(* IEC 61131-3 sources: codesys-mcp-toolkit/standalone-sync/sources_st/511_05, 13 files *)

(* ---- CLIENT_STATE.dut.st ---- *)
// @OBJECT_ID: 38106bf3-2e28-4407-a341-929dcc35d1f5
// @DECLARATION
// шаг состояния клиента
{attribute 'strict'}
TYPE CLIENT_STATE :
(
	CREATE	:=	 0,
	WAITING	:=	10,
	SEND	:=	20,
	RECEIVE :=  30
);
END_TYPE

(* ---- Coils.dut.st ---- *)
// @OBJECT_ID: 733d5e5a-4ad1-4a84-973a-cf97214e756a
// @DECLARATION
{attribute 'pack_mode' := '1'}
TYPE Coils :
STRUCT
// --- Режимы работы (команды из HMI) ---
xManualMode_Diazo   : BOOL;        // 1. Ручной режим Diazo
xManualMode_Soda    : BOOL;        // 2. Ручной режим Soda
xManualMode_Steam   : BOOL;        // 3. Ручной режим Steam
// --- Управление водой имитатором ---
xWaterValve_AutoMode : BOOL;       // 4. TRUE=Автоматический режим, FALSE=Ручной
xWaterValve_HmiOpen  : BOOL;       // 5. Открытие по кнопке из HMI (в ручном режиме)
xWaterValve_AutoReq  : BOOL;       // 6. Запрос на открытие от автоматики
// --- Сигналы запуска ---
xWaterStart          : BOOL;       // 7. Запуск дозы воды из HMI
xStartHeating_511    : BOOL;       // 8. Запуск прогрева
// --- Сигналы и статусы стадии промывки (Cascade Drain) ---
xStartCoupling_511   : BOOL;       // 9. Запуск с HMI: признак запуска стадии промывки
xCouplingActive_511  : BOOL;       // 10. Статус для HMI: признак "работа идет"
xCouplingDone_511    : BOOL;       // 11. Статус для HMI: признак "успешно готово"
// --- Режим удержания температуры ---
xKeepTempHeating_511 : BOOL;       // 12. TRUE = удержание температуры после нагрева, FALSE = разовый нагрев
// --- Служебные ---
PLC_READ             : BOOL := TRUE; // 13. Флаг чтения PLC
END_STRUCT
END_TYPE

(* ---- HoldingRegs.dut.st ---- *)
// @OBJECT_ID: e939cef4-c06c-4a02-a15a-aa924dd4400b
// @DECLARATION
{attribute 'pack_mode' := '4'}
TYPE HoldingRegs :
STRUCT
// =============================================================
// Модули M7–M9 (MDS AO-2UI) - Управление клапанами (Выходы 4-20мА)
// =============================================================

// --- Управление запорно-регулирующими клапанами (задание 0..100%) ---
AO1_CmdValveDiazo   : REAL;    // 101. Управление клапаном диазосоединения
AO2_CmdValveSoda    : REAL;    // 103. Управление клапаном едкого натра 14%
AO3_CmdValveSteam   : REAL;    // 105. Управление клапаном пара 6 ати

// --- Уставки с панели (ручной режим) ---
rValveManSet_Diazo  : REAL := 0.0;    // 107. Уставка с панели: Диазо
rValveManSet_Soda   : REAL := 0.0;    // 109. Уставка с панели: Сода
rValveManSet_Steam  : REAL := 0.0;    // 111. Уставка с панели: Пар

// --- Переменные для автоматического управления (выходы ПИД-регуляторов) ---
rAutoSet_Diazo      : REAL;           // 113. Выход ПИД расхода диазо
rAutoSet_Soda       : REAL;           // 115. Выход ПИД расхода соды
rAutoSet_Steam      : REAL;           // 117. Выход ПИД расхода пара

// --- Технологические уставки ---
rWaterDose          : REAL := 5.0;    // 119. Заданная доза воды, м³ (5 кубов)
rSetTempApp511      : REAL := 86.0;   // 121. Уставка температуры
rSetFlowDiazo_511   : REAL;           // 123. Уставка мгновенного расхода диазосоединения (до 19 м³/ч)
rSetPh_511          : REAL;           // 125. Целевая уставка pH (9.5..12 ед.)

// --- Настройки алгоритма опустошения емкости (для наладчика) ---
rZeroFlowThreshold_511 : REAL := 0.2; // 127. Порог падения расхода диазо (м³/ч), ниже которого считаем, что емкость пуста
uiEmptyDelaySec_511    : UINT := 20;  // 129. Задержка фиксации пустого трубопровода (сек)

// --- Настройки ПИД-регуляторов (для наладки контуров с HMI) ---
rKp_Diazo_511        : REAL := 1.0;   // 131. Пропорциональный коэффициент контура расхода диазосоединения
rTn_Diazo_511        : REAL := 5.0;   // 133. Время интегрирования контура расхода диазосоединения (сек)
rKp_pH_511           : REAL := 2.0;   // 135. Пропорциональный коэффициент контура pH
rTn_pH_511           : REAL := 10.0;  // 137. Время интегрирования контура pH (сек)
rKp_Steam_511        : REAL := 2.0;   // 139. Пропорциональный коэффициент контура пара (нагрева)
rTn_Steam_511        : REAL := 15.0;  // 141. Время интегрирования контура пара (сек)
rTv_Steam_511        : REAL := 0.0;   // 143. Время дифференцирования контура пара (сек)

END_STRUCT
END_TYPE

(* ---- InputRegs.dut.st ---- *)
// @OBJECT_ID: e329769f-e235-4ed6-8989-e7d305dd0344
// @DECLARATION
{attribute 'pack_mode' := '4'}
TYPE InputRegs :
STRUCT
	COILS : DINT := 0;
	INPUTS: DINT := 0;
	HOLDINGS: DINT := 0;
	INPUTREGS: DINT := 0;

  // МОДУЛЬ АНАЛОГОВЫХ ВХОДОВ (AI)
  	{region M1_K3_AI_10_08_00 }
    // =========================================================================
    // Первые 3 канала: Сигнализация положений (% открытия) клапанов [1, 2]
    (* adr 9 *)  rPosValveDiazo  : REAL; // Канал 1: Обратная связь клапана диазосоединения
    (* adr 11 *) rPosValveSoda   : REAL; // Канал 2: Обратная связь клапана едкого натра 14%
    (* adr 13 *) rPosValveSteam  : REAL; // Канал 3: Обратная связь клапана пара

    // Канал 4: рН-метр
    (* adr 15 *) rPhApp511       : REAL; // Канал 4: Показания pH-метра аппарата 511 (диапазон 9,5..12 ед.)
			{endregion}

	{region M5_MDS_3RTD_1 }
	(* adr 17 *) rTempApp511     : REAL; // Температура в аппарате 511 (до 100 С°)

   	{endregion}

	{region tenzo tv006c }
	(* adr 19 *) WE_1            : REAL;
	(* adr 21 *) WE_2            : REAL;

   	{endregion}

	{region tenzo ELMER }

	(* adr 23 *) IR_FlowSoda   : REAL; // Текущий расход щелочи , л/мин (или м3/ч)
	(* adr 25 *) IR_TotalSoda   : REAL; // Накопленный объем щелочи, л (или м3)
	(* adr 27 *) IR_FlowWater     : REAL; // Текущий расход воды, л/мин (или м3/ч)
	(* adr 29 *) IR_TotalWater   : REAL; // Накопленный объем воды, л (или м3)

    // Выходные сигналы загрузки воды
	(* adr  31*)   rWaterLoaded   : REAL;    // Сколько воды загружено, м³
	(* adr 32*)    rWaterStatus   : REAL;    // Статус загрузки воды: 0=IDLE 1=RUNNING 2=DONE 3=ABORTED

	(* adr  33*)  IR_FlowDiazo   : REAL; // Текущий мгновенный расход диазосоединения (м3/ч) [3]
	(* adr  35*)  IR_TotalDiazo   : REAL; // Текущий расход диазосоединения, л/мин (или м3/ч)

	(* adr  37*)  rDizoStatus   : REAL; // Текущий расход диазосоединения, л/мин (или м3/ч)

	(* adr  39*) rDiazoLoaded   : REAL; // Текущий расход диазосоединения, л/мин (или м3/ч)
rTimeLeft_511:REAL ;///Оставшиеся секунды при падении расхода
	 rStateCode_511:REAL;//

   	{endregion}

END_STRUCT
END_TYPE

(* ---- Inputs.dut.st ---- *)
// @OBJECT_ID: a5893dca-19fc-4f6d-bdfc-9d37b1592804
// @DECLARATION
{attribute 'pack_mode' := '1'}
TYPE Inputs :
STRUCT
			// =============================================================
			// Модуль M11 (MDS DIO-16BD) - Статусы насосов (Дискретные входы)
			// =============================================================
			{region M11 - MDS DIO-16BD (Статусы насосов)}

    // Выходная переменная на физическое реле/соленоид
    xWaterValve_Out     : BOOL;  // 1 канал ФЕ
	xWaterValve_SQH :BOOL;
	xWaterValve_SQL   :BOOL;
			{endregion}
END_STRUCT
END_TYPE

(* ---- GVL.gvl.st ---- *)
// @OBJECT_ID: 3f8320a4-dc77-4c55-9b52-3e7e3f19e8e0
// @DECLARATION
{attribute 'qualified_only'}

VAR_GLOBAL

	gInputRegs	:	InputRegs;
	gHoldingRegs	:	HoldingRegs;
	gInputs	:	Inputs;
	gCoils	:	Coils;
    // =========================================================================
    // АНАЛОГОВЫЕ ВХОДЫ (Опрос датчиков)
    // =========================================================================
    rPressPump207v      : REAL; // Давление насоса мембранного 207в (0.5..6 кгс/см2)
    rTempApp511         : REAL; // Температура реакционной среды в аппарате 511 (до 100 °C)
    rPhApp511           : REAL; // Показания pH-метра аппарата 511 (9.5..12 ед.)

	WE_1_s:WORD;
	WE_1_f:WORD;

	WE_2_s:WORD;
	WE_2_f:WORD;

	sStateStr_511:string(255);

    // =========================================================================
    // СЧЕТЧИКИ И РАСХОДОМЕРЫ (Опрос текущего расхода и накопленного объема)
    // =========================================================================
    rFlowDiazo          : REAL; // Текущий расход диазосоединения (м3/ч)
    rTotalDiazo         : REAL; // Накопленный объем диазосоединения (м3)

    rFlowSoda           : REAL; // Текущий расход едкого натра 14% (м3/ч)
    rTotalSoda          : REAL; // Накопленный объем едкого натра 14% (м3)

    rFlowWater          : REAL; // Текущий расход воды артезианской/деминерализованной (м3/ч)
    rTotalWater         : REAL; // Накопленный объем воды / счетчик дозы (м3)

    // =========================================================================
    // СИГНАЛЫ СОСТОЯНИЯ КЛАПАНОВ (Входы обратной связи)
    // =========================================================================
    rPosValveDiazo      : REAL; // Сигнализация положения (% открытия) клапана диазосоединения
    rPosValveSoda       : REAL; // Сигнализация положения (% открытия) клапана едкого натра
    rPosValveSteam      : REAL; // Сигнализация положения (% открытия) клапана пара

    xStsValveWaterOpen  : BOOL; // Сигнализатор положения отсечного пневмокрана воды - ОТКРЫТ
    xStsValveWaterClose : BOOL; // Сигнализатор положения отсечного пневмокрана воды - ЗАКРЫТ

    // =========================================================================
    // АНАЛОГОВЫЕ И ДИСКРЕТНЫЕ ВЫХОДЫ (Управление исполнительными механизмами)
    // =========================================================================
    rCmdValveDiazo  AT  %QW0    : WORD; // Управление регулирующим клапаном диазосоединения (0..100%)
    rCmdValveSoda   AT  %QW1    : WORD; // Управление регулирующим клапаном едкого натра (0..100%)
    rCmdValveSteam  AT  %QW2    : WORD; // Управление регулирующим клапаном пара для поддержания температуры (0..100%)
    xCmdValveWater      : BOOL; // Дискретное управление отсечным пневмокраном воды (закрытие при достижении дозы)

    // =========================================================================
    // ПЕРЕМЕННЫЕ HMI / СЕНСОРНОЙ ПАНЕЛИ (Уставки и задания)
    // =========================================================================
    rSpTempApp511       : REAL; // Задание поддерживаемой температуры в аппарате (до 100 °C)
    rSpFlowDiazo        : REAL; // Задание необходимого расхода диазосоединения (до 19 м3/ч)
    rSpFlowSoda         : REAL; // Задание необходимого расхода едкого натра (до 7.35 м3/ч)
    rSpDoseWater        : REAL; // Задание необходимой дозы воды (до 7.35 м3/ч)

    // Переменные для алгоритма дозирования щелочи
    rSpPhLow            : REAL := 9.2; // Нижний порог pH для увеличения открытия клапана щелочи
    rSpPhHigh           : REAL := 9.7; // Верхний порог pH для уменьшения открытия клапана щелочи
    rSpPhTargetMatch    : REAL := 9.6; // Порог pH для открытия клапана щелочи на стадии "сочетания"
    rSpPhTargetClose    : REAL := 9.5; // Порог pH для закрытия клапана щелочи
MDS_3RTD_1_start_ad : POINTER TO ARRAY[0..10] OF WORD;;
END_VAR

(* ---- PVL.gvl.st ---- *)
// @OBJECT_ID: d4c88051-2adb-4578-9e31-dd205f936f9c
// @DECLARATION
{attribute 'qualified_only'}
VAR_GLOBAL PERSISTENT RETAIN
	rHoldingRegs: HoldingRegs;
END_VAR

(* ---- FC_Write_AO.func.st ---- *)
// @OBJECT_ID: 58eab0a1-f642-4bbd-ba35-3845d9d3886b
// @DECLARATION
FUNCTION FC_Write_AO : BOOL
VAR_INPUT
    VAL_IN  : REAL;    // Входное значение (например, от ПИД 0..1000)

    pOutput : POINTER TO ARRAY[0..1] OF WORD; // Адрес физических регистров модуля
END_VAR
VAR
    TMP     : REAL;
    dwValue : DWORD;
	    X1      : REAL:=0;    // Мин. вход (например, 0)
    X2      : REAL:=100;    // Макс. вход (например, 1000)
    Y1      : REAL:=4;    // Мин. ток (например, 4.0)
    Y2      : REAL:=20;    // Макс. ток (например, 20.0)
END_VAR

// @IMPLEMENTATION

// 1. Проверка на нулевой указатель и деление на ноль
IF pOutput = 0 OR (X2 = X1) THEN
    FC_Write_AO := FALSE;
    RETURN;
END_IF;

// 2. Линейное масштабирование (из входного диапазона в 4..20мА)
TMP := (Y2 - Y1) / (X2 - X1) * (VAL_IN - X1) + Y1;

// 3. Преобразование REAL во внутреннее битовое представление DWORD
dwValue := OSCAT_BASIC.REAL_TO_DW(TMP);

// 4. Запись напрямую в память по указателю (разбивка на 2 WORD)
// В ПЛК Абак обычно старшее слово идет первым (зависит от настроек модуля)
pOutput^[0] := OSCAT_BASIC.WORD_OF_DWORD(dwValue, 1); // High Word
pOutput^[1] := OSCAT_BASIC.WORD_OF_DWORD(dwValue, 0); // Low Word

FC_Write_AO := TRUE;

(* ---- FC_Write_AO_CDAB.func.st ---- *)
// @OBJECT_ID: c5f4f6d9-aef8-4f24-80c9-f3d975bafcdd
// @DECLARATION
FUNCTION FC_Write_AO_CDAB : BOOL
VAR_INPUT
    rValIn   : REAL;    // Входная уставка (0..100)
    pOutput  : POINTER TO ARRAY[0..1] OF WORD;
    rInMin   : REAL;
    rInMax   : REAL;
    rOutMin  : REAL;
    rOutMax  : REAL;
END_VAR
VAR
    rScaled  : REAL;
    dwRaw    : DWORD;
	dwCDAB: DWORD;
    pReal    : POINTER TO DWORD;
END_VAR

// @IMPLEMENTATION
// 1. Линейное масштабирование (Scale)
// Формула: Out = ((In - InMin) * (OutMax - OutMin) / (InMax - InMin)) + OutMin
IF (rInMax <> rInMin) THEN
    rScaled := ((rValIn - rInMin) * (rOutMax - rOutMin) / (rInMax - rInMin)) + rOutMin;
ELSE
    rScaled := rOutMin;
END_IF

// 2. Получаем битовое представление REAL как DWORD
pReal := ADR(rScaled);
dwRaw := pReal^;

// 3. Перепаковка в формат CDAB
// Исходный (ABCD): [Byte3][Byte2][Byte1][Byte0]
// Формат CDAB:     [Byte1][Byte0][Byte3][Byte2]
// То есть меняем местами слова (WORD)

dwCDAB := ROL(dwRaw, 16); // Простейший способ поменять слова местами

// 4. Запись результата по указателю
IF pOutput <> 0 THEN
    pOutput^[1] := DWORD_TO_WORD(dwCDAB AND 16#FFFF);        // Младшее слово CDAB (бывшее старшее AB)
    pOutput^[0] := DWORD_TO_WORD(SHR(dwCDAB, 16));           // Старшее слово CDAB (бывшее младшее CD)
    FC_Write_AO_CDAB := TRUE;
ELSE
    FC_Write_AO_CDAB := FALSE;
END_IF

(* ---- FB_AI.fb.st ---- *)
// @OBJECT_ID: 3f0a8be8-2f33-46cf-a2ab-090e0d72fc51
// @DECLARATION
FUNCTION_BLOCK FB_AI
VAR_INPUT
	F_WORD_IN : WORD;
	S_WORD_IN : WORD;
	X1 : REAL:=4;
	Y1 : REAL:=0;
	X2 : REAL:=20;
	Y2 : REAL:=100;
	RANGE_CONV:BOOL:=TRUE;
END_VAR
VAR
	TMP:REAL;
END_VAR
VAR_OUTPUT
	VAL_OUT : REAL;
END_VAR

// @IMPLEMENTATION
TMP := OSCAT_BASIC.DW_TO_REAL(X:= OSCAT_BASIC.DWORD_OF_WORD(W1:= F_WORD_IN , W0:= S_WORD_IN ));
IF (RANGE_CONV)
THEN
	IF (TMP=9999 OR TMP=-9999 OR TMP=-7777 OR TMP=7777)
	THEN
		VAL_OUT :=  TMP;
	ELSE
		VAL_OUT :=  (Y2 - Y1) / (X2 - X1) * (TMP - X1) + Y1;
	END_IF

ELSE
	VAL_OUT :=  TMP;
END_IF

(* ---- FB_ModbusToFloatArray.fb.st ---- *)
// @OBJECT_ID: 8d81ca1b-e4d0-4e94-b201-9038cef709f6
// @DECLARATION
FUNCTION_BLOCK FB_ModbusToFloatArray
VAR_INPUT
    aDataIn : ARRAY [0..219] OF WORD; // Входной массив (до 120 регистров)
    iQty    : INT := 1;               // Количество FLOAT переменных для обработки (макс 60)
    iMode   : INT := 1;               // Режим: 0=1234, 1=3412 (частый), 2=2143, 3=4321
END_VAR
VAR_OUTPUT
    aDataOut : ARRAY [0..119] OF REAL; // Выходной массив
    xError   : BOOL;                  // Флаг ошибки (если iQty > 60)
END_VAR
VAR
    i : INT;
    uConverter : U_WordToReal;
    wLow : WORD;
    wHigh : WORD;
    wTemp1 : WORD;
    wTemp2 : WORD;
END_VAR

// @IMPLEMENTATION

// Сброс ошибки
xError := FALSE;

// Защита от выхода за пределы массива
IF iQty < 1 OR iQty > 120 THEN
    xError := TRUE;
    RETURN;
END_IF

// Основной цикл
FOR i := 0 TO (iQty - 1) DO

    // Получаем пару регистров из массива
    // i*2 - это начало пары (0, 2, 4...)
    wTemp1 := aDataIn[i * 2];     // Первый регистр пары
    wTemp2 := aDataIn[(i * 2) + 1]; // Второй регистр пары

    CASE iMode OF
        // ---------------------------------------------------------
        // Mode 0: 1234 (Big Endian)
        // Порядок: [HighWord] [LowWord]
        // ---------------------------------------------------------
        0:
            wHigh := wTemp1;
            wLow  := wTemp2;

        // ---------------------------------------------------------
        // Mode 1: 3412 (Middle Little / Word Swap) -> САМЫЙ ЧАСТЫЙ для Modbus
        // Порядок: [LowWord] [HighWord]
        // Регистры меняются местами, байты внутри - нет.
        // ---------------------------------------------------------
        1:
            wHigh := wTemp2;
            wLow  := wTemp1;

        // ---------------------------------------------------------
        // Mode 2: 2143 (Middle Big / Byte Swap)
        // Порядок: [HighWord swapped] [LowWord swapped]
        // Байты меняются местами внутри каждого слова.
        // ---------------------------------------------------------
        2:
            wHigh := ROL(wTemp1, 8); // Меняем байты местами
            wLow  := ROL(wTemp2, 8);

        // ---------------------------------------------------------
        // Mode 3: 4321 (Little Endian)
        // Порядок: [LowWord swapped] [HighWord swapped]
        // Полный разворот: меняются и слова, и байты.
        // ---------------------------------------------------------
        3:
            wHigh := ROL(wTemp2, 8);
            wLow  := ROL(wTemp1, 8);

        ELSE
            // По умолчанию используем 3412 (как самый популярный)
            wHigh := wTemp2;
            wLow  := wTemp1;
    END_CASE

    // Сборка DWORD из двух слов
    // Сдвигаем старшее слово на 16 бит влево и добавляем младшее
    uConverter.dwValue := SHL(WORD_TO_DWORD(wHigh), 16) OR WORD_TO_DWORD(wLow);

    // Запись результата в выходной массив
    aDataOut[i] := uConverter.rValue;

END_FOR

(* ---- ASK_prg.prg.st ---- *)
// @OBJECT_ID: 34a98575-253b-42d3-9455-2cb10a7687ff
// @DECLARATION
PROGRAM ASK_prg
VAR
Exatract:	FB_ModbusToFloatArray;
pt : POINTER TO  ARRAY [0..5] OF WORD  ;

//M1_K3_AI_10_08_00 AT %IW58: ARRAY [0..7] OF WORD ;

buff_abak: ARRAY [0..219] OF WORD ;
buff_MDS: ARRAY [0..219] OF WORD ;
buffR_1: ARRAY [0..119] OF REAL ;
start_ad_mds3rtd:INT:=0;
swap_mds3rtd:INT:=6;
start_ad_mds_8UId:INT:=18;
swap_mds_8UI:INT:=16;

AI: FB_AI;

	Info : __SYSTEM.VAR_INFO;

    pAddress : POINTER TO BYTE;
	adress:UDINT;
END_VAR

// @IMPLEMENTATION
//берем  с модуля  M1_K3_AI_10_08_00 значения  и  копируем в промежуточный буфер
SysMemCpy(ADR(buff_abak), ADR( %IW0), 8 * SIZEOF(WORD));

//берем  с модуля  MDS_3RTD_1  значения  и  копируем в промежуточный буфер
SysMemCpy(ADR(buff_MDS), ADR( %IW57), 6 * SIZEOF(WORD));

//берем  с  терминала  tv 006
SysMemCpy(ADR(buff_MDS[swap_mds3rtd]), ADR( %IW53), 2* SIZEOF(WORD));

//берем  с  терминала  tv 006
SysMemCpy(ADR(buff_MDS[swap_mds3rtd+2]), ADR( %IW55), 2* SIZEOF(WORD));

Exatract(aDataIn:=buff_MDS,aDataOut=>buffR_1,IQty:=65,iMode:=1);

// 3. Маппинг (Присвоение значений переменным структуры)
// -------------------------------------------------------------

// === Модуль M1 () ===
GVL.gInputRegs. rPosValveDiazo  := AIToFloat(buff_abak[0],0,100); //
GVL.gInputRegs.rPosValveSoda  := AIToFloat(buff_abak[1],0,100); //
GVL.gInputRegs.rPosValveSteam  := AIToFloat(buff_abak[2],0,100); //
GVL.gInputRegs.rPhApp511  := AIToFloat(buff_abak[4],0,14); //

// === Модуль M5 () ===

GVL.gInputRegs.rTempApp511  :=buffR_1[0];// TT 511
//GVL.gInputRegs.rTempApp511  :=FC_ModbusToRealSwapped(wWord1 := buff_MDS[0], wWord2 := buff_MDS[1]);
// === Модуль M2 () ===
GVL.rCmdValveDiazo := FloatToAI(gvl.gHoldingRegs.AO1_CmdValveDiazo);

GVL.rCmdValveSoda := FloatToAI(gvl.gHoldingRegs.AO2_CmdValveSoda);

GVL.rCmdValveSteam := FloatToAI(gvl.gHoldingRegs.AO3_CmdValveSteam);

// === Модуль M5 (Индексы 0..2) ===
//GVL.gInputRegs.rTempApp511   := buffR_1[0]; // TT 511

//// === весы  tenzo  M1 ===

	//AI(F_WORD_IN:= gvl.WE_1_f, S_WORD_IN:= gvl.WE_1_s, RANGE_CONV:=FALSE, VAL_OUT=> GVL.gInputRegs.WE_1);
GVL.gInputRegs.WE_1:=buffR_1[3];
GVL.gInputRegs.WE_2:=buffR_1[4];
//// === весы  tenzo  M2 ===
//AI(F_WORD_IN:= gvl.WE_2_f, S_WORD_IN:= gvl.WE_2_s, RANGE_CONV:=TRUE, VAL_OUT=> GVL.gInputRegs.WE_2);

(* ---- PLC_PRG.prg.st ---- *)
// @OBJECT_ID: 4c4237aa-22c6-43a4-ae1d-3ca0359860c2
// @DECLARATION
PROGRAM PLC_PRG // Antigravity Sync Test
VAR
    fbElemerREM         : fbElemerREM;

    (* Переменные из вкладки Modbus Generic Serial Slave I/O Mapping *)
    Hmi_Flow_Regs    AT %IW67  : ARRAY[0..1] OF WORD; (* Канал 0 (Мгновенный расход) *)
    Hmi_Volume_Regs  AT %IW63  : ARRAY[0..3] OF WORD; (* Канал 1 (Накопленный объем) *)
    xModbusCommError    : BOOL;                 (* Системный флаг ошибки связи с прибором *)
    xHmiResetCmd        : BOOL;                 (* Сигнал сброса сумматора с HMI-панели *)

    (* Выходные очищенные технологические переменные *)
    rCurrentFlowRate    : REAL;                 (* Мгновенный расход в систему, куб.м/ч *)
    lrAccumulatedVol    : LREAL;                (* Точный накопленный объем, куб.м *)
    sOperatorMessage    : STRING(255);          (* Сообщение для текстовой строки на панели *)

    fbWater             : FB_WaterLoading;      (* Наш исправленный ФБ дозирования *)

    // ============================================================
    // ПЕРЕМЕННЫЕ ДЛЯ ТЕСТИРОВАНИЯ И СИМУЛЯЦИИ СУММАТОРА
    // ============================================================
    xSimEnable          : BOOL := FALSE;        (* Включить режим симуляции (True = подмена датчиков) *)
    rSimFlowSpeed       : REAL := 20.0;         (* Скорость потока при открытом клапане, куб.м/ч *)
    rSimTotalStorage    : REAL := 125.45;       (* Внутренний виртуальный накопительный счетчик куб.м *)

    fbSimClock          : TON;                  (* Генератор тактов времени для подсчета объема *)
    rDeltaVolume        : REAL;                 (* Математический шаг приращения за 1 такт *)
    // ============================================================
END_VAR

// @IMPLEMENTATION
// ================================================================
// 1. ЧТЕНИЕ РЕАЛЬНЫХ ДАННЫХ ИЗ ПОЛЕВЫХ ПРИБОРОВ
// ================================================================
gvl.gInputRegs.IR_TotalSoda := F_ElemerREM_Volume(pBuf := ADR(%IW65));
gvl.gInputRegs.IR_FlowSoda  := F_ElemerREM_Flow(pBuf := ADR(%IW69));
gvl.gInputRegs.rTempApp511  := F_GetReal_BADC(pBuf := ADR(%IW57));

// ================================================================
// 2. ДИНАМИЧЕСКИЙ СИМУЛЯТОР РАСХОДОМЕРА ВОДЫ
// ================================================================
// Тактовый генератор: срабатывает каждые 100 мс (0.1 секунды) для плавности хода счета
fbSimClock(IN := xSimEnable AND NOT fbSimClock.Q, PT := T#100ms);

IF xSimEnable THEN
    // ЕСЛИ СИМУЛЯЦИЯ ВКЛЮЧЕНА:

    // Имитируем поведение потока в зависимости от команды на клапан
    IF gvl.gCoils.xWaterValve_AutoReq THEN
        // Клапан открыт автоматикой -> задаем симуляционный расход
        gvl.gInputRegs.IR_FlowWater := rSimFlowSpeed;

        // Расчет приращения сумматора за 100мс: (куб.м/ч * 0.1с) / 3600с
        IF fbSimClock.Q THEN
            rDeltaVolume := (rSimFlowSpeed * 0.1) / 3600.0;
            rSimTotalStorage := rSimTotalStorage + rDeltaVolume;
        END_IF;
    ELSE
        // Клапан закрыт -> поток прекращается
        gvl.gInputRegs.IR_FlowWater := 0.0;
    END_IF;

    // ПОДМЕНЯЕМ значение сумматора результатом симуляции для ФБ дозирования
    gvl.gInputRegs.IR_TotalWater := rSimTotalStorage;

ELSE
    // ЕСЛИ СИМУЛЯЦИЯ ВЫКЛЮЧЕНА (РАБОЧИЙ РЕЖИМ):

    // Читаем физический прибор с адреса %IW71 и %IW75
    gvl.gInputRegs.IR_TotalWater := F_ElemerREM_Volume(pBuf := ADR(%IW71));
    gvl.gInputRegs.IR_FlowWater  := F_ElemerREM_Flow(pBuf := ADR(%IW75));

    // Мягко синхронизируем симулятор, чтобы при включении тумблера счет не прыгал назад/вперед
    rSimTotalStorage := gvl.gInputRegs.IR_TotalWater;
END_IF;

// ================================================================
// 3. ВЫЗОВ И ПРОВЕРКА ФУНКЦИОНАЛЬНОГО БЛОКА ЗАГРУЗКИ ВОДЫ
// ================================================================
fbWater(
    rTotalVolume := gvl.gInputRegs.IR_TotalWater,        // Сюда идет либо физический объем, либо симуляция
    rDose        := gvl.gHoldingRegs.rWaterDose,         // Заданная уставка дозы (куб.м)
    rDeadband    := 0.05,                                // Упреждение закрытия (0.05 куб.м)
    xStart       := gvl.gCoils.xWaterStart,              // Команда Старт/Стоп
    xMode        := gvl.gCoils.xWaterValve_AutoMode,     // Флаг режима АВТО клапана
    xAutoControl := gvl.gCoils.xWaterValve_AutoReq       // Управление клапаном (выход на открытие)
);

    gvl.gInputRegs.rWaterLoaded:=fbWater.rLoaded;
    gvl.gInputRegs.rWaterStatus:=fbWater.rStatus;
